// TIA Portal V20 export
DATA_BLOCK "InstProfinetDeviceDiag_x2"   // DB209
AUTHOR : Siemens Digital Industries
FAMILY : LAF
VERSION : 1.2
// stored: AssignedProDiagFB ProDiag, InstanceOfName LAF_ProfinetDevDiag, InstanceOfType FB
"LAF_ProfinetDevDiag"
   // VAR_INPUT
   //    plantIdentifier { ExternalAccessible := 'False'; ExternalVisible := 'False'; ExternalWritable := 'False'} : WString[24] := WSTRING#'';
   //    textListId { ExternalAccessible := 'False'; ExternalVisible := 'False'; ExternalWritable := 'False'} : Int := 0;
   //    localProfinetSystem { ExternalAccessible := 'False'; ExternalVisible := 'False'; ExternalWritable := 'False'} : HW_IOSYSTEM := 0;
   //    firstCycle { ExternalAccessible := 'False'; ExternalVisible := 'False'; ExternalWritable := 'False'} : Bool := FALSE;
   //    maxDevicesDiag { ExternalAccessible := 'False'; ExternalVisible := 'False'; ExternalWritable := 'False'} : DInt := 0;
   //    maxModulesDiag { ExternalAccessible := 'False'; ExternalVisible := 'False'; ExternalWritable := 'False'} : DInt := 0;
   //    ackAlarms { ExternalAccessible := 'False'; ExternalVisible := 'False'; ExternalWritable := 'False'} : Bool := FALSE;
   //    hideAlarmMask { ExternalAccessible := 'False'; ExternalVisible := 'False'; ExternalWritable := 'False'} : Word := 16#0000;
   // END_VAR
   // VAR_OUTPUT
   //    generalAlarm { ExternalAccessible := 'False'; ExternalVisible := 'False'; ExternalWritable := 'False'} : Bool := FALSE;
   //    deviceFaulty { ExternalAccessible := 'False'; ExternalVisible := 'False'; ExternalWritable := 'False'} : Bool := FALSE;
   //    deviceProblem { ExternalAccessible := 'False'; ExternalVisible := 'False'; ExternalWritable := 'False'} : Bool := FALSE;
   //    deviceDeactivated { ExternalAccessible := 'False'; ExternalVisible := 'False'; ExternalWritable := 'False'} : Bool := FALSE;
   //    deviceNotPresent { ExternalAccessible := 'False'; ExternalVisible := 'False'; ExternalWritable := 'False'} : Bool := FALSE;
   // END_VAR
   // VAR_IN_OUT
   //    interfaceDevDiag : "LAF_typeDevDiagInterface";
   // END_VAR
   // VAR
   //    statDevDiagInternal { ExternalAccessible := 'False'; ExternalVisible := 'False'; ExternalWritable := 'False'} : "LAF_typeDevDiagInternal";
   //    statCnt1ShotGetName { ExternalAccessible := 'False'; ExternalVisible := 'False'; ExternalWritable := 'False'} : DInt := 1;
   //    statCnt1ShotGeo2Log { ExternalAccessible := 'False'; ExternalVisible := 'False'; ExternalWritable := 'False'} : DInt := 1;
   //    statCnt1ShotGetImDat { ExternalAccessible := 'False'; ExternalVisible := 'False'; ExternalWritable := 'False'} : DInt := 1;
   //    statCntCyclDevState { ExternalAccessible := 'False'; ExternalVisible := 'False'; ExternalWritable := 'False'} : DInt := 1;
   //    statCntCyclState { ExternalAccessible := 'False'; ExternalVisible := 'False'; ExternalWritable := 'False'} : DInt := 1;
   //    statCntCyclModulState { ExternalAccessible := 'False'; ExternalVisible := 'False'; ExternalWritable := 'False'} : DInt := 1;
   //    statCntCyclGetDiag { ExternalAccessible := 'False'; ExternalVisible := 'False'; ExternalWritable := 'False'} : DInt := 1;
   //    statBusy { ExternalAccessible := 'False'; ExternalVisible := 'False'; ExternalWritable := 'False'} : "LAF_typeDevDiagStateInstruct";
   //    statDone { ExternalAccessible := 'False'; ExternalVisible := 'False'; ExternalWritable := 'False'} : "LAF_typeDevDiagStateInstruct";
   //    statOtherInstruct { ExternalAccessible := 'False'; ExternalVisible := 'False'; ExternalWritable := 'False'} : "LAF_typeDevDiagInstruct";
   //    instGetName { ExternalAccessible := 'False'; ExternalVisible := 'False'; ExternalWritable := 'False'} : Get_Name;
   //    statGetNameDat { ExternalAccessible := 'False'; ExternalVisible := 'False'; ExternalWritable := 'False'} : String[24] := '';
   //    statGetNameErrorStatus { ExternalAccessible := 'False'; ExternalVisible := 'False'; ExternalWritable := 'False'} : Word := 16#0000;
   //    statGetNameErrorDevCycle { ExternalAccessible := 'False'; ExternalVisible := 'False'; ExternalWritable := 'False'} : DInt := 0;
   //    instGetImData { ExternalAccessible := 'False'; ExternalVisible := 'False'; ExternalWritable := 'False'} : Get_IM_Data;
   //    statIm0Data { ExternalAccessible := 'False'; ExternalVisible := 'False'; ExternalWritable := 'False'} : IM0_Data;
   //    statGetImDatErrorStatus { ExternalAccessible := 'False'; ExternalVisible := 'False'; ExternalWritable := 'False'} : Word := 16#0000;
   //    statGetImDatErrorCycle { ExternalAccessible := 'False'; ExternalVisible := 'False'; ExternalWritable := 'False'} : DInt := 0;
   //    statAlarm { ExternalAccessible := 'False'; ExternalVisible := 'False'; ExternalWritable := 'False'} : "LAF_typeDevDiagAlarm";
   //    statHideAlarm { ExternalAccessible := 'False'; ExternalVisible := 'False'; ExternalWritable := 'False'} : "LAF_typeDevDiagAlarm";
   //    statRisPushbutton { ExternalAccessible := 'False'; ExternalVisible := 'False'; ExternalWritable := 'False'} : "LAF_typeDevDiagRisEdge";
   //    statErrorText { ExternalAccessible := 'False'; ExternalVisible := 'False'; ExternalWritable := 'False'} : String[24] := 'No Device Name readable';
   //    stat8CharError { ExternalAccessible := 'False'; ExternalVisible := 'False'; ExternalWritable := 'False'} : String[8] := '????????';
   //    statAlarmNo { ExternalAccessible := 'False'; ExternalVisible := 'False'; ExternalWritable := 'False'} : Array[0..23] of UInt;
   // END_VAR
BEGIN
   statDevDiagInternal.localProfinetSystem := 0;
   statDevDiagInternal.maxDevices := 0;
   statDevDiagInternal.maxModules := 0;
   statDevDiagInternal.numberDevices.configured := 0;
   statDevDiagInternal.numberDevices.notPresent := 0;
   statDevDiagInternal.numberDevices.deactivated := 0;
   statDevDiagInternal.numberDevices.faulty := 0;
   statDevDiagInternal.numberDevices.problem := 0;
   statDevDiagInternal.hwAddress[0..256].hwtype2 := 0;
   statDevDiagInternal.hwAddress[0..256].hwtype5 := 0;
   statDevDiagInternal.hwAddress[0..256].hwtype5If := 0;
   statBusy.getName := FALSE;
   statBusy.geo2Log := FALSE;
   statBusy.moduleStates := FALSE;
   statBusy.getDiag := FALSE;
   statBusy.getImData := FALSE;
   statDone.getName := FALSE;
   statDone.geo2Log := FALSE;
   statDone.moduleStates := FALSE;
   statDone.getDiag := FALSE;
   statDone.getImData := FALSE;
   statOtherInstruct.log2GeoLaddr := 0;
   statOtherInstruct.log2GeoRetVal := 0;
   statOtherInstruct.log2Geo.HWTYPE := 0;
   statOtherInstruct.log2Geo.AREA := 0;
   statOtherInstruct.log2Geo.IOSYSTEM := 0;
   statOtherInstruct.log2Geo.STATION := 0;
   statOtherInstruct.log2Geo.SLOT := 0;
   statOtherInstruct.log2Geo.SUBSLOT := 0;
   statOtherInstruct.devStateMode1.laddr := 0;
   statOtherInstruct.devStateMode1.mode := 0;
   statOtherInstruct.devStateMode1.retVal := 0;
   statOtherInstruct.devStateMode1.state[0..1024] := FALSE;
   statOtherInstruct.devStateMode2.laddr := 0;
   statOtherInstruct.devStateMode2.mode := 0;
   statOtherInstruct.devStateMode2.retVal := 0;
   statOtherInstruct.devStateMode2.state[0..1024] := FALSE;
   statOtherInstruct.devStateMode3.laddr := 0;
   statOtherInstruct.devStateMode3.mode := 0;
   statOtherInstruct.devStateMode3.retVal := 0;
   statOtherInstruct.devStateMode3.state[0..1024] := FALSE;
   statOtherInstruct.devStateMode4.laddr := 0;
   statOtherInstruct.devStateMode4.mode := 0;
   statOtherInstruct.devStateMode4.retVal := 0;
   statOtherInstruct.devStateMode4.state[0..1024] := FALSE;
   statOtherInstruct.devStateMode5.laddr := 0;
   statOtherInstruct.devStateMode5.mode := 0;
   statOtherInstruct.devStateMode5.retVal := 0;
   statOtherInstruct.devStateMode5.state[0..1024] := FALSE;
   statOtherInstruct.geo2LogLaddr := 0;
   statOtherInstruct.geo2LogRetVal := 0;
   statOtherInstruct.geo2Log.HWTYPE := 0;
   statOtherInstruct.geo2Log.AREA := 0;
   statOtherInstruct.geo2Log.IOSYSTEM := 0;
   statOtherInstruct.geo2Log.STATION := 0;
   statOtherInstruct.geo2Log.SLOT := 0;
   statOtherInstruct.geo2Log.SUBSLOT := 0;
   statOtherInstruct.moduleStateMode2.laddr := 0;
   statOtherInstruct.moduleStateMode2.mode := 0;
   statOtherInstruct.moduleStateMode2.retVal := 0;
   statOtherInstruct.moduleStateMode2.state[0..127] := FALSE;
   statOtherInstruct.moduleStateMode5.laddr := 0;
   statOtherInstruct.moduleStateMode5.mode := 0;
   statOtherInstruct.moduleStateMode5.retVal := 0;
   statOtherInstruct.moduleStateMode5.state[0..127] := FALSE;
   statOtherInstruct.getDiag.mode := 0;
   statOtherInstruct.getDiag.laddr := 0;
   statOtherInstruct.getDiag.retVal := 0;
   statOtherInstruct.getDiag.cntDiag := 0;
   statOtherInstruct.getDiag.diagDataMode0 := 16#0000_0000;
   statOtherInstruct.getDiag.diagDataMode1.MaintainanceState := 16#0000_0000;
   statOtherInstruct.getDiag.diagDataMode1.ComponentStateDetail := 16#0000_0000;
   statOtherInstruct.getDiag.diagDataMode1.OwnState := 0;
   statOtherInstruct.getDiag.diagDataMode1.IOState := 16#0000;
   statOtherInstruct.getDiag.diagDataMode1.OperatingState := 0;
   statOtherInstruct.getDiag.diagDataMode2.SubordinateState := 0;
   statOtherInstruct.getDiag.diagDataMode2.SubordinateIOState := 16#0000;
   statOtherInstruct.getDiag.diagDataMode2.DNNmode := 16#0000;
   statOtherInstruct.getDiag.detailData := 0;
   instGetName.LADDR := 0;
   instGetName.STATION_NR := 0;
   instGetName.DONE := FALSE;
   instGetName.BUSY := FALSE;
   instGetName.ERROR := FALSE;
   instGetName.LEN := 0;
   instGetName.STATUS := 16#0000;
   instGetName.BusyState := 16#0000;
   instGetImData.LADDR := 0;
   instGetImData.IM_TYPE := 0;
   instGetImData.DONE := FALSE;
   instGetImData.BUSY := FALSE;
   instGetImData.ERROR := FALSE;
   instGetImData.STATUS := 16#0000;
   instGetImData.sdw_GetAttrID := 16#0000_0000;
   instGetImData.sdw_GetAttrAID := 16#0000_0000;
   instGetImData.sdi_SfcLen := 0;
   instGetImData.sb_useGetMultiAttr := FALSE;
   instGetImData.sui_GetMultiAttrACount := 0;
   instGetImData.sa_GetMultiAttrPathLens[0] := 0;
   instGetImData.sa_GetMultiAttrPaths[0..2] := 0;
   instGetImData.sa_GetMultiAttrResultLens[0] := 0;
   instGetImData.sa_GetMultiAttrResult := '';
   instGetImData.sb_SfcValid := FALSE;
   instGetImData.sb_SfcERROR := FALSE;
   instGetImData.sw_SfcStatus := 16#0000;
   instGetImData.sa_SfcData[0..64] := 16#00;
   instGetImData.sudi_arraylength := 0;
   instGetImData.sudi_datatype := 0;
   instGetImData.sui_imdataLen := 0;
   instGetImData.sui_imdataLen_netto := 54;
   instGetImData.si_index := 0;
   instGetImData.sb_SfcLocked := FALSE;
   instGetImData.pw_TemporaryWord := 16#0000;
   instGetImData.pa_DataByte[0..53] := 16#00;
   instGetImData.pa_DataChar[0..53] := ' ';
   instGetImData.pa_TemporaryCharArray[0..19] := ' ';
   instGetImData.p_DataUDT.Manufacturer_ID := 0;
   instGetImData.p_DataUDT.Order_ID := '';
   instGetImData.p_DataUDT.Serial_Number := '';
   instGetImData.p_DataUDT.Hardware_Revision := 0;
   instGetImData.p_DataUDT.Software_Revision."Type" := ' ';
   instGetImData.p_DataUDT.Software_Revision.Functional := 0;
   instGetImData.p_DataUDT.Software_Revision.Bugfix := 0;
   instGetImData.p_DataUDT.Software_Revision.Internal := 0;
   instGetImData.p_DataUDT.Revision_Counter := 0;
   instGetImData.p_DataUDT.Profile_ID := 0;
   instGetImData.p_DataUDT.Profile_Specific_Type := 0;
   instGetImData.p_DataUDT.IM_Version := 16#0000;
   instGetImData.p_DataUDT.IM_Supported := 16#0000;
   statIm0Data.Manufacturer_ID := 0;
   statIm0Data.Order_ID := '';
   statIm0Data.Serial_Number := '';
   statIm0Data.Hardware_Revision := 0;
   statIm0Data.Software_Revision."Type" := ' ';
   statIm0Data.Software_Revision.Functional := 0;
   statIm0Data.Software_Revision.Bugfix := 0;
   statIm0Data.Software_Revision.Internal := 0;
   statIm0Data.Revision_Counter := 0;
   statIm0Data.Profile_ID := 0;
   statIm0Data.Profile_Specific_Type := 0;
   statIm0Data.IM_Version := 16#0000;
   statIm0Data.IM_Supported := 16#0000;
   statAlarm.invalidValueMaxDevices := FALSE;
   statAlarm.invalidValueMaxModules := FALSE;
   statAlarm.invalidAddressLog2Geo := FALSE;
   statAlarm.errorReadDeviceStates := FALSE;
   statAlarm.deviceFaulty := FALSE;
   statAlarm.deviceProblem := FALSE;
   statAlarm.deviceDeactivated := FALSE;
   statAlarm.deviceNotPresent := FALSE;
   statAlarm.deviceNetworkError := FALSE;
   statAlarm.deviceMaintRequired := FALSE;
   statAlarm.deviceMaintDemanded := FALSE;
   statAlarm.spare11 := FALSE;
   statAlarm.spare12 := FALSE;
   statAlarm.spare13 := FALSE;
   statAlarm.spare14 := FALSE;
   statAlarm.spare15 := FALSE;
   statHideAlarm.invalidValueMaxDevices := FALSE;
   statHideAlarm.invalidValueMaxModules := FALSE;
   statHideAlarm.invalidAddressLog2Geo := FALSE;
   statHideAlarm.errorReadDeviceStates := FALSE;
   statHideAlarm.deviceFaulty := FALSE;
   statHideAlarm.deviceProblem := FALSE;
   statHideAlarm.deviceDeactivated := FALSE;
   statHideAlarm.deviceNotPresent := FALSE;
   statHideAlarm.deviceNetworkError := FALSE;
   statHideAlarm.deviceMaintRequired := FALSE;
   statHideAlarm.deviceMaintDemanded := FALSE;
   statHideAlarm.spare11 := FALSE;
   statHideAlarm.spare12 := FALSE;
   statHideAlarm.spare13 := FALSE;
   statHideAlarm.spare14 := FALSE;
   statHideAlarm.spare15 := FALSE;
   statRisPushbutton.risEdgeManualReadAll := FALSE;
   statRisPushbutton.posPulseManualReadAll := FALSE;
   statRisPushbutton.risEdgeResetAll := FALSE;
   statRisPushbutton.posPulseResetAll := FALSE;
   statRisPushbutton.risEdgeQuitAlarms := FALSE;
   statRisPushbutton.posPulseQuitAlarms := FALSE;
   statAlarmNo[0] := 0;
   statAlarmNo[1] := 1;
   statAlarmNo[2] := 2;
   statAlarmNo[3] := 3;
   statAlarmNo[4] := 4;
   statAlarmNo[5] := 5;
   statAlarmNo[6] := 6;
   statAlarmNo[7] := 7;
   statAlarmNo[8] := 8;
   statAlarmNo[9] := 9;
   statAlarmNo[10] := 10;
   statAlarmNo[11] := 11;
   statAlarmNo[12] := 12;
   statAlarmNo[13] := 13;
   statAlarmNo[14] := 14;
   statAlarmNo[15] := 15;
   statAlarmNo[16] := 16;
   statAlarmNo[17] := 17;
   statAlarmNo[18] := 18;
   statAlarmNo[19] := 19;
   statAlarmNo[20] := 20;
   statAlarmNo[21] := 21;
   statAlarmNo[22] := 22;
   statAlarmNo[23] := 23;
END_DATA_BLOCK
